PROGRAM Main
VAR
END_VAR

END_PROGRAM

(* stored: Version 1.1.0.1, ProductVersion 3.1.4024.12
   POU Main: Id {fda65918-0421-47aa-928e-2b446155a782}, SpecialFunc None *)
